TYPE ES_T6 :
	STRUCT
		Alarm			:ES_ALARM;
	
		S1_rt			:R_TRIG;	
		S1_letto		:BOOL;
	END_STRUCT
END_TYPE

(* stored: Version 1.1.0.1, ProductVersion 3.1.4022.12
   DUT ES_T6: Id {249f8325-7ffe-47ae-8be9-3731b48e61ae} *)
